Universal Robots PolyScope program: d02_unplug.urp

Program d02_unplug (installation=default directory=/programs createdIn=5.9.1.1031110 lastSavedIn=5.9.1.1031110 robotSerialNumber=20195501059)
Calibrated DH parameters: a=[0.000146, -0.418764, -0.053981, 0.000058, -0.000023, 0]; d=[0.162545, 37.319448, -206.067439, 168.881546, 0.09955, 0.099464]; alpha=[1.57004, -0.001979, 0.002304, 1.570607, -1.57066, 0]; deltaTheta=[0, -0.174616, -1.258233, 1.432844, -0.000001, 0]
Robot Program (runOnlyOnce=true)
  MoveL speed 250 mm/s, acceleration 1200 mm/s^2 (useActiveTCP=true) feature=Base
    Waypoint Waypoint (Variable): variable(featureName=d02_plug_p)
    URCap Gripper (Robotiq_Grippers, Robotiq Inc.) dataModel(position=100.0, force=100.0, speed=100.0, positionInDouble=100.0, forceInDouble=100.0, speedInDouble=100.0, slaveIds=[9], blocking=false)
    MoveDirectionNode (selectedDirection=ZPlus toolParams=0.02, 0.8) feature=Joint_6_name
      Until TOOL_CONTACT_DETECTION (allowActions=true retraction=0.001 decelerationAcceleration=3 decelerationAngularAcceleration=34.906585)
        URCap Gripper (Robotiq_Grippers, Robotiq Inc.) dataModel(position=65.0, force=100.0, speed=100.0, positionInDouble=65.0, forceInDouble=100.0, speedInDouble=100.0, slaveIds=[9], blocking=true)
        MoveDirectionNode (selectedDirection=ZPlus toolParams=0.05, 0.8) feature=Joint_6_name
          Until DISTANCE (allowActions=false deceleration=3 distanceNodeType=STOP) Distance=0.02; motionParameters(blendRadius=0)
        URCap Gripper (Robotiq_Grippers, Robotiq Inc.) dataModel(position=100.0, force=100.0, speed=100.0, positionInDouble=100.0, forceInDouble=100.0, speedInDouble=100.0, slaveIds=[9], blocking=true)
        MoveL speed 25 mm/s, acceleration 1200 mm/s^2 (useActiveTCP=true) feature=Base
          Waypoint Pull (Relative): relativeFromPosition TCP in base x=108.075 y=-582.031 z=19.139 mm, rx=-2.2457 ry=-2.1683 rz=0.0242 rad; joints [88.128, -64.848, 105.271, -130.26, 268.593, 90.173] deg; TCP offset x=0 y=0 z=174 mm, rx=0 ry=0 rz=0 rad; TCP in base x=109.536 y=-542.231 z=19.13 mm, rx=-2.2458 ry=-2.1682 rz=0.0241 rad; joints [88.149, -69.075, 111.89, -132.649, 268.605, 90.202] deg
      Until DISTANCE (allowActions=true deceleration=3 distanceNodeType=STOP) Distance=0.02; motionParameters(blendRadius=0)
        Waypoint Waypoint (Variable): variable(featureName=d02_plug_p)
